FUNCTION Buffer_Layout_Set_SInt_Array : UINT
VAR_INPUT
END_VAR
VAR
END_VAR

END_FUNCTION

(* stored: Version 1.1.0.1, ProductVersion 3.1.4024.10
   POU Buffer_Layout_Set_SInt_Array: Id {a2ce18ac-13e9-44be-8f20-8526f15a1cab}, SpecialFunc None *)
